(* basic NC axis ctrl *)
FUNCTION_BLOCK FB_MC2_BasicAxisCtrl
VAR_INPUT
	bEnable				: BOOL;		(* set TRUE to enable axis and drive *)
	bReset				: BOOL;		(* set TRUE to reset axis from ERROR conditionh *)
	bEnableRevDir		: BOOL;		(* set TRUE to allow motion in reverse direction *)
	fOverride			: LREAL;	(* max axis output in % *)
END_VAR
VAR_IN_OUT
	stParamSet			: ST_AxisParameterSet;	(* axis parameter set *)
	stAxis				: AXIS_REF;	(* axis structure *)
END_VAR
VAR_OUTPUT
	bInitOK				: BOOL;		(* TRUE = parameter set read OK *)
	bEnabled			: BOOL;		(* TRUE = axis enabled *)
	bActive				: BOOL;		(* TRUE = axis running *)
	bRunningFwd			: BOOL;		(* TRUE = axis running forwards *)
	bRunningRev			: BOOL;		(* TRUE = axis running reverse *)
	bCalibrated			: BOOL;		(* TRUE = axis has been referenced *)
	bAxisError			: BOOL;		(* TRUE = NC axis error *)
	nAxisErrorID		: UDINT;	(* NC axis error code *)
	fActPos				: LREAL;	(* actual absolute position *)
	fModuloPos			: LREAL;	(* actual modulo position *)
	fActVelo			: LREAL;	(* actual velocity *)
END_VAR
VAR
	fbReadParamSet		: MC_ReadParameterSet;
	fbInitOK			: RS;
	fbReadStatus		: MC_ReadStatus;
	fbPower				: MC_Power;

	fbReqReset			: RS;
	fbReset				: MC_Reset;
	fbEnableOffEvent	: F_TRIG;
	fbReqUnlock			: RS;
	fbUnlock			: MC_GearOut;
	bSyncPulse: BOOL;
END_VAR
(*
-------------------------------------------------------------------------------------------------
Date		Version	Author	Comments
-------------------------------------------------------------------------------------------------
30/01/2015	3.00.00	PB		Phasing introduced to prevent cyclic commands being issued at the same time from multiple axes
							MC_ReadParameterSet now phased across 1s using FB_SquareWave, AxisID as offset value giving 1ms phase between axes
							MC_Reset and MC_GearOut now phased across 50ms using FB_SquareWave, AxisID / 8 as offset value allowing 8 commands per 1ms cycle

-------------------------------------------------------------------------------------------------
21/03/2012	1.09.00	PB		Renamed FB_MC2_BasicAxisCtrl
25/03/2011	1.06.02	PB		Bug fix - Oriented Stop using MC_MoveModulo now called when when axis has stopped accelerating
							NOTE:  awaiting response from Beckhoff regarding MC_MoveModulo aborting if called while axis is accelerating
							NOTE:  awaiting response from Beckhoff regarding NC axis crash if MC_Halt is used to cancel axis acceleration
							Oriented Stop now also used to bring axis to stop if error occurs with MC_MoveVelocity commands
							FastStop still used to bring axis to immediate stop if error occurs with MC_Jog
24/01/2011	1.06.01	PB		FastStop now called if any internal motion command fails
13/10/2010	1.05.01	PB		If fSetVelo = 0 units/sec, axis will now come to stop
							NC axis will not accept velocity ref <0.001 unit/sec, so NC axis will also stop
23/09/2010	1.03.02	PB		bInitOK flag will now be cancelled if error occurs with axis parameter set
11/08/2010	1.03.01	PB		Oriented stop now works when running backwards
06/07/2010	1.02.01	PB		Oriented stop modified to improve reliability, MC_MoveVelocity (added in V1.01.01) removed
							Fast Stop is triggered if MC_MoveModulo stop cannot be achieved
							MC_GearOut added to automatically unlock axis if enable signal is lost
28/06/2010	1.01.02	PB		Axis parameter set now refreshed every 1 sec
14/06/2010	1.01.01	PB		MC_MoveVelocity added before MC_MoveModulo to ensure new ramps are used for oriented stop
							If MC_MoveModulo fails or aborts for any reason, MC_Stop is called to ensure axis is stopped
05/02/2010	1.00.00	PB		Initial release

-------------------------------------------------------------------------------------------------
*)

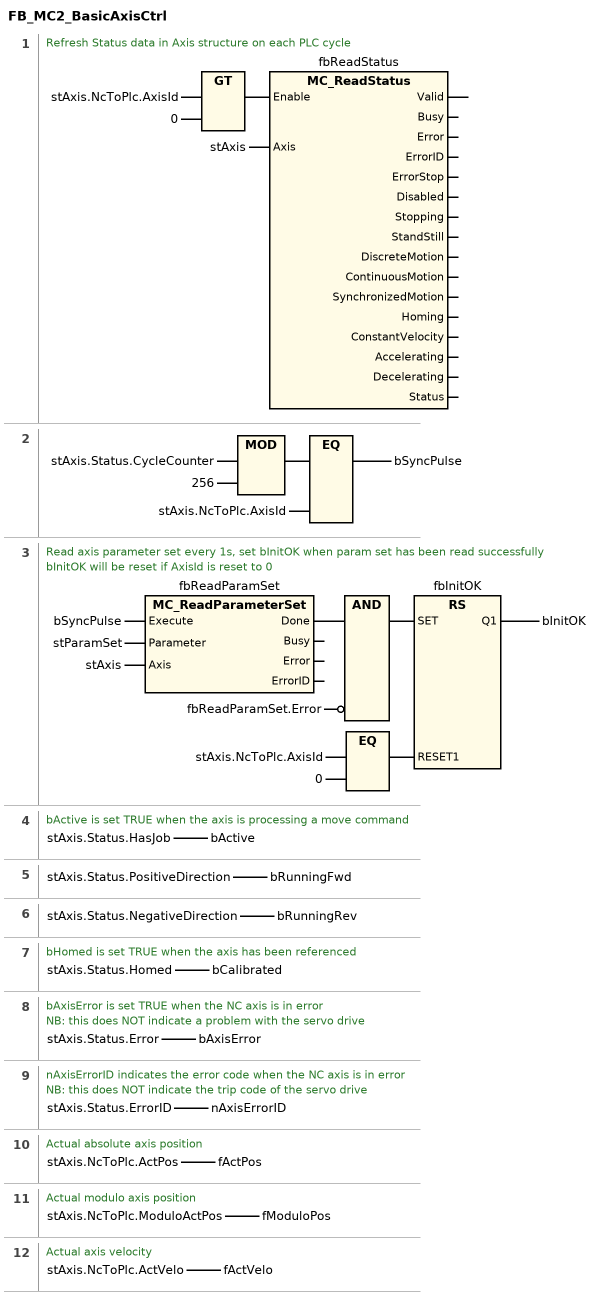
// NETWORK 1
// Refresh Status data in Axis structure on each PLC cycle
fbReadStatus(Enable := stAxis.NcToPlc.AxisId > 0, Axis := stAxis); // MC_ReadStatus

// NETWORK 2
bSyncPulse := stAxis.Status.CycleCounter MOD 256 = stAxis.NcToPlc.AxisId;

// NETWORK 3
// 					Read axis parameter set every 1s, set bInitOK when param set has been read successfully
// bInitOK will be reset if AxisId is reset to 0
//
fbReadParamSet(Execute := bSyncPulse, Parameter := stParamSet, Axis := stAxis); // MC_ReadParameterSet
fbInitOK(SET := fbReadParamSet.Done AND NOT fbReadParamSet.Error, RESET1 := stAxis.NcToPlc.AxisId = 0); // RS
bInitOK := fbInitOK.Q1;

// NETWORK 4
// bActive is set TRUE when the axis is processing a move command
bActive := stAxis.Status.HasJob;

// NETWORK 5
bRunningFwd := stAxis.Status.PositiveDirection;

// NETWORK 6
bRunningRev := stAxis.Status.NegativeDirection;

// NETWORK 7
// bHomed is set TRUE when the axis has been referenced
bCalibrated := stAxis.Status.Homed;

// NETWORK 8
// 					bAxisError is set TRUE when the NC axis is in error
// NB: this does NOT indicate a problem with the servo drive
//
bAxisError := stAxis.Status.Error;

// NETWORK 9
// 					nAxisErrorID indicates the error code when the NC axis is in error
// NB: this does NOT indicate the trip code of the servo drive
//
nAxisErrorID := stAxis.Status.ErrorID;

// NETWORK 10
// Actual absolute axis position
fActPos := stAxis.NcToPlc.ActPos;

// NETWORK 11
// Actual modulo axis position
fModuloPos := stAxis.NcToPlc.ModuloActPos;

// NETWORK 12
// Actual axis velocity
fActVelo := stAxis.NcToPlc.ActVelo;

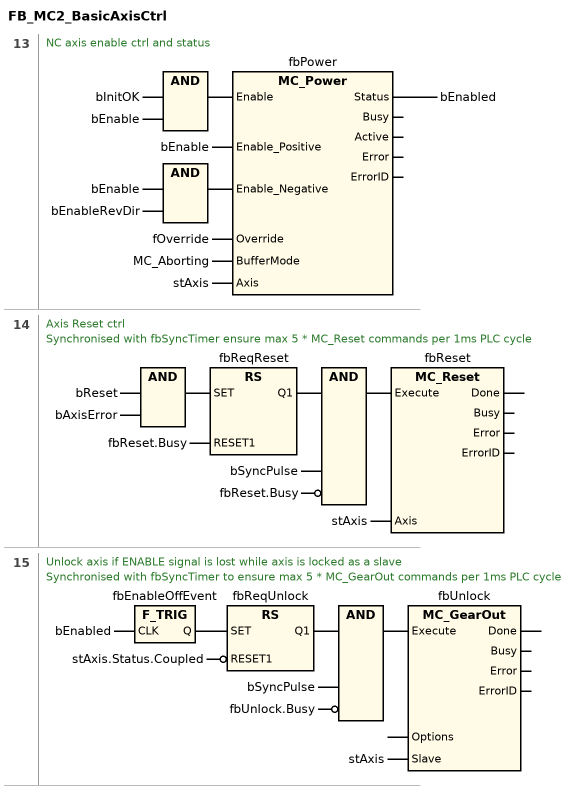
// NETWORK 13
// NC axis enable ctrl and status
fbPower(
    Enable := bInitOK AND bEnable,
    Enable_Positive := bEnable,
    Enable_Negative := bEnable AND bEnableRevDir,
    Override := fOverride,
    BufferMode := MC_Aborting,
    Axis := stAxis); // MC_Power
bEnabled := fbPower.Status;

// NETWORK 14
// 					Axis Reset ctrl
// Synchronised with fbSyncTimer ensure max 5 * MC_Reset commands per 1ms PLC cycle
//
fbReqReset(SET := bReset AND bAxisError, RESET1 := fbReset.Busy); // RS
fbReset(Execute := fbReqReset.Q1 AND bSyncPulse AND NOT fbReset.Busy, Axis := stAxis); // MC_Reset

// NETWORK 15
// 					Unlock axis if ENABLE signal is lost while axis is locked as a slave
// Synchronised with fbSyncTimer to ensure max 5 * MC_GearOut commands per 1ms PLC cycle
//
fbEnableOffEvent(CLK := bEnabled); // F_TRIG
fbReqUnlock(SET := fbEnableOffEvent.Q, RESET1 := NOT stAxis.Status.Coupled); // RS
fbUnlock(Execute := fbReqUnlock.Q1 AND bSyncPulse AND NOT fbUnlock.Busy, Slave := stAxis); // MC_GearOut

END_FUNCTION_BLOCK

(* stored: Version 1.1.0.1, ProductVersion 3.1.4024.15
   POU FB_MC2_BasicAxisCtrl: Id {ec4f0983-b831-468f-9701-189a3d336d27}, SpecialFunc None *)
